PROGRAM MAIN
VAR
	trigger : BOOL := TRUE;
	createGuid : FB_CreateGuid;
	guid : GUID;
	guidAsString : STRING;
END_VAR

IF NOT createGuid.bBusy AND trigger THEN	
	
	trigger := FALSE;
	createGuid(bExecute := FALSE);	
	createGuid(
			bExecute := TRUE,
			pGuidBuffer := ADR(guid),
			nGuidBufferSize := SIZEOF(guid));
			
ELSIF createGuid.bBusy THEN
	
	createGuid();	
	
END_IF

// The code abover this point does not require any further libraries.  
// ------------------------------------------------------------------
// The code below requires Tc2_Utilites

guidAsString := GUID_TO_STRING(guid);

END_PROGRAM

(* stored: Version 1.1.0.1, ProductVersion 3.1.4024.5
   POU MAIN: Id {dd60aeb8-b539-4862-864e-f793c1299126}, SpecialFunc None *)
